// TIA Portal V20 export
VAR_GLOBAL   // PLC tag table "PHMI"
   "BA030AZSD1PHMI.I[0]" AT %IW189 : Int;
   "BA030AZSD1PHMI.Q[0]" AT %QW189 : Int;
END_VAR
VAR_GLOBAL CONSTANT   // user constants
   "OB_Safety.ProDiagOB(1)" : OB_PCYCLE := 251;
   "OB_CyclicInterruptReceiveData(1)" : OB_Cyclic := 30;
   "OB_Safety.FOB_RTG1(1)" : OB_Cyclic := 123;
END_VAR
